{attribute 'hide'}
FUNCTION_BLOCK FileSystemEntry_Test EXTENDS TcUnit.FB_TestSuite

EmptyPathReturnsExpected();
PathAppendsBackslashIfRequired();

METHOD EmptyPathReturnsExpected
VAR
	expected : FilePath;
	actual : FilePath;
	mockFileSystemEntry : Mock_FilesystemEntry('');
END_VAR
TEST('EmptyPathReturnsExpected');

// @TEST-FIXTURE

// @TEST-RUN
expected := '.\';
actual := mockFileSystemEntry.Path;

// @TEST-ASSSERT
AssertEquals_STRING(Expected := expected, Actual := actual, Message := 'Empty path did not return expected');

TEST_FINISHED();
END_METHOD

METHOD PathAppendsBackslashIfRequired
VAR
	expected : FilePath;
	actual : FilePath;
	mockFileSystemEntry : Mock_FilesystemEntry('C:\temp');
END_VAR
TEST('PathAppendsBackslashIfRequired');

// @TEST-FIXTURE

// @TEST-RUN
expected := 'C:\temp\';
actual := mockFileSystemEntry.Path;

// @TEST-ASSSERT
AssertEquals_STRING(Expected := expected, Actual := actual, Message := 'Path did not return expected');

TEST_FINISHED();
END_METHOD

END_FUNCTION_BLOCK

(* stored: Version 1.1.0.1, ProductVersion 3.1.4024.9
   POU FileSystemEntry_Test: Id {5cb30f18-e69e-4fe1-9679-47172b385adc}, SpecialFunc None
   Method EmptyPathReturnsExpected: Id {1514409c-d8c6-4d6c-b823-fcbdfc54c49c}
   Method PathAppendsBackslashIfRequired: Id {c54ca597-8631-4e86-af61-2c4568128ee1} *)
